// TIA Portal V20 export
DATA_BLOCK "DB_OPC_Machine"   // DB15
{ S7_Optimized_Access := 'TRUE' }
// stored: MemoryReserve 100
   VAR
      Parts : Struct
         Out : Struct
            Station1 : Struct
               LoaderDrilled : SInt;
               LoaderUndrilled : SInt;
               ShuttleDrilled : SInt;
               ShuttleUndrilled : SInt;
               WorkClamp : SInt;
            END_STRUCT;
         END_STRUCT;
      END_STRUCT;
      State : Struct
         Current : Struct
            CanLockDoor : Bool;
            CanUnlockDoor : Bool;
            CncMode : Byte;
            LoadingMode : Byte;
            IsDoorLocked : Bool;
            IsEmptying : Bool;
            IsInitialized : Bool;
            IsRunning : Bool;
            MachineOverride : Byte;
         END_STRUCT;
         Requests : Struct
            LoadingMode : Struct
               RequestChangeMode : Bool;
               TargetMode : Byte;
            END_STRUCT;
            RequestLockDoor : Bool;
            RequestStartAuto : Bool;
            RequestStartEmptying : Bool;
            RequestStopAuto : Bool;
            RequestStopEmptying : Bool;
            RequestUnlockDoor : Bool;
         END_STRUCT;
      END_STRUCT;
   END_VAR
   VAR RETAIN
      Parameters : Struct
         GasAssistSetPoint : Real;
         CoolingVentilatorSetpoint : Real;
         TemperatureCoolingSetpoint : Real;
         BlowingSetpoint : Real;
         Shuttle1Enable : "UDT_BoolEnable";
         Shuttle2Enable { S7_SetPoint := 'True'} : "UDT_BoolEnable";
         ConsecutiveBwIn { S7_SetPoint := 'True'} : Int;
         Sequence : Struct
            Shuttle1 : Struct
               Main : Int;
               ShuttleInt : Int;
               ShuttleExt : Int;
               ControlIn : Int;
               ControlOut : Int;
               Blowing : Int;
               IntLoadUnload : Int;
               ExtLoadUnload : Int;
               BwLoadUnload : Int;
               BwControlIn : Int;
               ActControlIn : Int;
               ActControlOut : Int;
               ActBwControlIn : Int;
            END_STRUCT;
            Shuttle2 : Struct
               Main : Int;
               ShuttleInt : Int;
               ShuttleExt : Int;
               ControlIn : Int;
               ControlOut : Int;
               Blowing : Int;
               IntLoadUnload : Int;
               ExtLoadUnload : Int;
               BwLoadUnload : Int;
               BwControlIn : Int;
               ActControlIn : Int;
               ActControlOut : Int;
               ActBwControlIn : Int;
            END_STRUCT;
            Fixture : Struct
               Blowing : Int;
               Loading : Int;
               Unloading : Int;
               V_Init : Int;
               W_Init : Int;
            END_STRUCT;
         END_STRUCT;
         Presence : Struct
            Shuttle1UndrilledPart : Bool;
            Shuttle1UndrilledBw : Bool;
            Shuttle1DrilledPart : Bool;
            Shuttle1DrilledBw : Bool;
            Shuttle2UndrilledPart : Bool;
            Shuttle2UndrilledBw : Bool;
            Shuttle2DrilledPart : Bool;
            Shuttle2DrilledBw : Bool;
            GripperUndrilledPart : Bool;
            GripperUndrilledBw : Bool;
            GripperDrilledPart : Bool;
            GripperDrilledBw : Bool;
            FixtureUndrilledPart : Bool;
            FixtureUndrilledBw : Bool;
            FixtureDrilledPart : Bool;
            FixtureDrilledBw : Bool;
         END_STRUCT;
      END_STRUCT;
   END_VAR
BEGIN
END_DATA_BLOCK
